(* LS Electric XG5000 project: test *)
(* PLC LSPLC *)
(* module base 0 slot 0: 입출력 모듈:XGH-DT4A (DC 24V 입력, 트랜지스터 출력 32점 ) *)
VAR_GLOBAL
    INST : TON;
END_VAR

PROGRAM NewProgram (* task: 스캔 프로그램 *)
VAR
    BCDOUT : WORD;
    DOG : TIME;
    IN1 : BOOL;
    IN2 : BOOL;
    input : BOOL;
    INST1 : TOF;
    INST2 : TP;
    INST3 : TON_UINT;
    LAMP2 : BOOL;
    MOTOR1 : BOOL;
    MOTOR2 : BOOL;
    MOTOR3 : BOOL;
    MOVEIN : INT;
    MOVEOUT : INT;
    on : INT;
    ONOFF : BOOL;
    out : BOOL;
    OUT1 : BOOL;
    output : BOOL;
    OUTPUT123 : BOOL;
    PB0 : BOOL;
    PB1 : BOOL;
    PLUSE : BOOL;
    PRATICE1 : BOOL;
    PULSE : BOOL;
    SOU1 : BOOL;
    SSUN : UINT;
    SUM : INT;
    T1 : TON;
    T2 : TOF;
    T2_SWITCH : BOOL;
    T3 : TP;
    T4 : TON_UINT;
    TON_UNIT : BOOL;
    x0 : BOOL;
    x1 : BOOL;
    x10 : BOOL;
    x11 : BOOL;
    x12 : BOOL;
    x2 : BOOL;
    x3 : BOOL;
    x4 : BOOL;
    x5 : BOOL;
    x6 : BOOL;
    x7 : BOOL;
    x8 : BOOL;
    x9 : BOOL;
    Y0 : BOOL;
    Y1 : BOOL;
    Y2 : BOOL;
    Y3 : BOOL;
    Y4 : BOOL;
    결과1 : INT;
    결과1_R : REAL;
    숫자1 : INT;
    숫자1_R : REAL;
    조명 : BOOL;
END_VAR
VAR_EXTERNAL
    INST : TON;
END_VAR
VAR
    _e1 : R_TRIG;
    _e2 : R_TRIG;
    _e3 : R_TRIG;
    _e4 : R_TRIG;
    _e5 : R_TRIG;
END_VAR

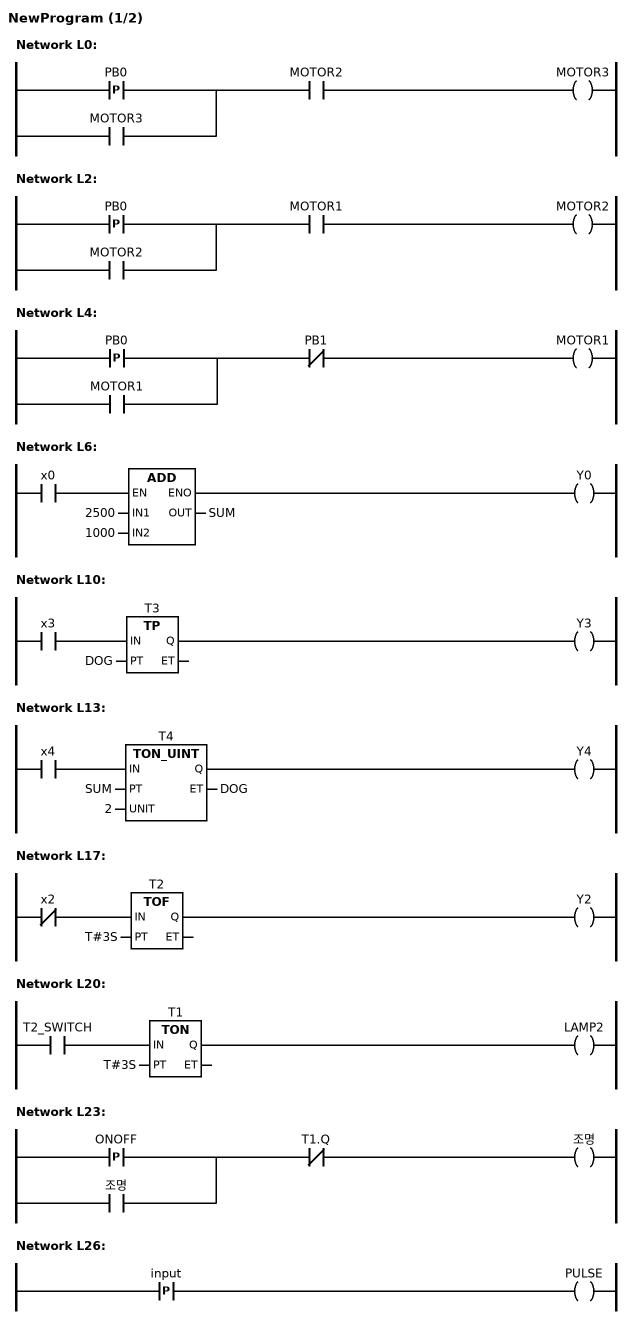
(* Rung L0 *)
_e1(CLK := PB0);
MOTOR3 := (_e1.Q OR MOTOR3) AND MOTOR2;
(* Rung L2 *)
_e2(CLK := PB0);
MOTOR2 := (_e2.Q OR MOTOR2) AND MOTOR1;
(* Rung L4 *)
_e3(CLK := PB0);
MOTOR1 := (_e3.Q OR MOTOR1) AND NOT PB1;
(* Rung L6 *)
IF x0 THEN SUM := 2500 + 1000; END_IF;
Y0 := x0;
(* Rung L10 *)
T3(IN := x3, PT := DOG);
Y3 := T3.Q;
(* Rung L13 *)
T4(IN := x4, PT := SUM, UNIT := 2, ET => DOG);
Y4 := T4.Q;
(* Rung L17 *)
T2(IN := NOT x2, PT := T#3S);
Y2 := T2.Q;
(* Rung L20 *)
T1(IN := T2_SWITCH, PT := T#3S);
LAMP2 := T1.Q;
(* Rung L23 *)
_e4(CLK := ONOFF);
조명 := (_e4.Q OR 조명) AND NOT T1.Q;
(* Rung L26 *)
_e5(CLK := input);
PULSE := _e5.Q;

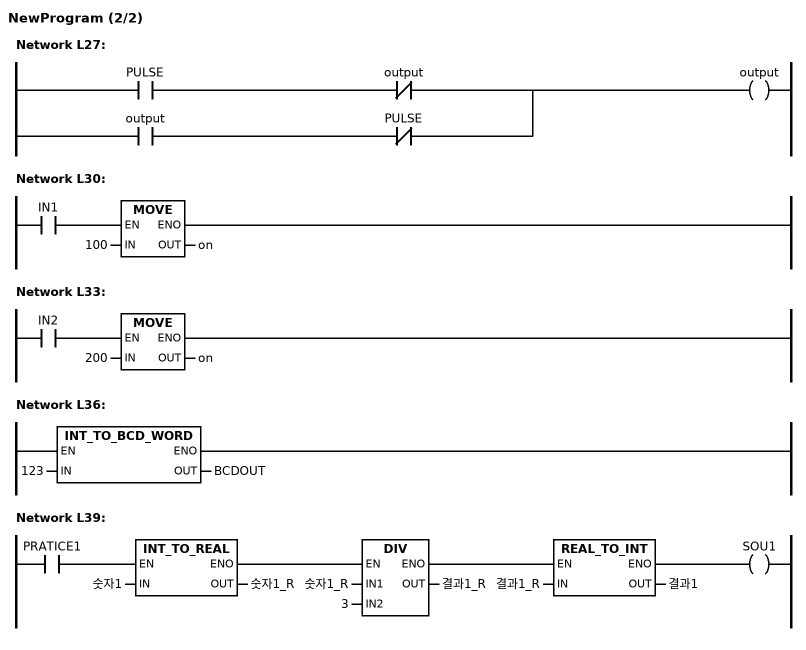
(* Rung L27 *)
output := (PULSE AND NOT output) OR (output AND NOT PULSE);
(* Rung L30 *)
IF IN1 THEN on := 100; END_IF;
(* Rung L33 *)
IF IN2 THEN on := 200; END_IF;
(* Rung L36 *)
BCDOUT := INT_TO_BCD_WORD(123);
(* Rung L39 *)
IF PRATICE1 THEN
    숫자1_R := INT_TO_REAL(숫자1);
    결과1_R := 숫자1_R / 3;
    결과1 := REAL_TO_INT(결과1_R);
END_IF;
SOU1 := PRATICE1;
END_PROGRAM